TYPE MoverSort :
STRUCT
	MoverNumber 	: UDINT;
	TrackID  		: PlanarTrackOTCID;
	MoverPos 		: LREAL;
	MoverTrackNr 	: UDINT;
END_STRUCT
END_TYPE

(* stored: Version 1.1.0.1, ProductVersion 3.1.4026.8
   DUT MoverSort: Id {2ab215a1-e1dc-4200-b2c9-e846d3f77aee} *)
